// LS Electric XG5000 project: 통신 테스트
// PLC LSPLC
// module base 0 slot 0: 입출력 모듈:XBC-DR32H (DC 24V 입력, 릴레이 출력 32점)

PROGRAM NewProgram (task: 스캔 프로그램)

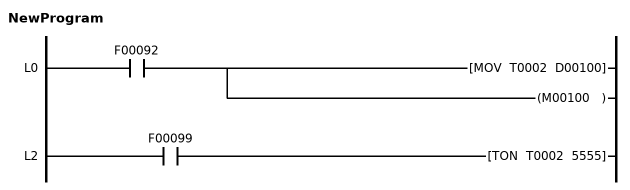
; L0
LOAD      F00092
MOV       T0002 D00100
OUT       M00100
; L2
LOAD      F00099
TON       T0002 5555